Omron CX-Programmer project НовыйПроект (CX-Programmer 9.52)

# PLC testPLC: CP1L-E EM

## Global symbols (name address type ; comment)
input1 0.00 BOOL  ; адр 1 тумблера
out1 100.00 BOOL  ; диск выход 100.00

## Program НоваяЗадача1 (cyclic task 0)
Local symbols
input2 W0.01 BOOL  ; вирт кнопка панели
out2 W100.03 BOOL  ; 88
out3 W0.06 BOOL  ; jjlll

### Section Сегмент1

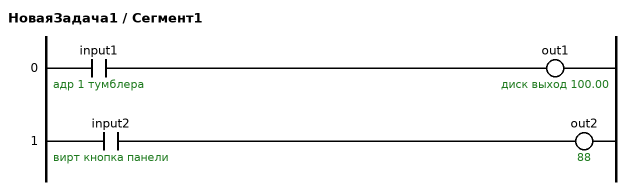
; rung 0
LD input1  ; адр 1 тумблера
OUT out1  ; диск выход 100.00
; rung 1
LD input2  ; вирт кнопка панели
OUT out2  ; 88

### Section END
; rung 0
END(001)